// Mitsubishi GX Works2 project: 14   PLC: FX2N/FX2NC

PROGRAM MAIN
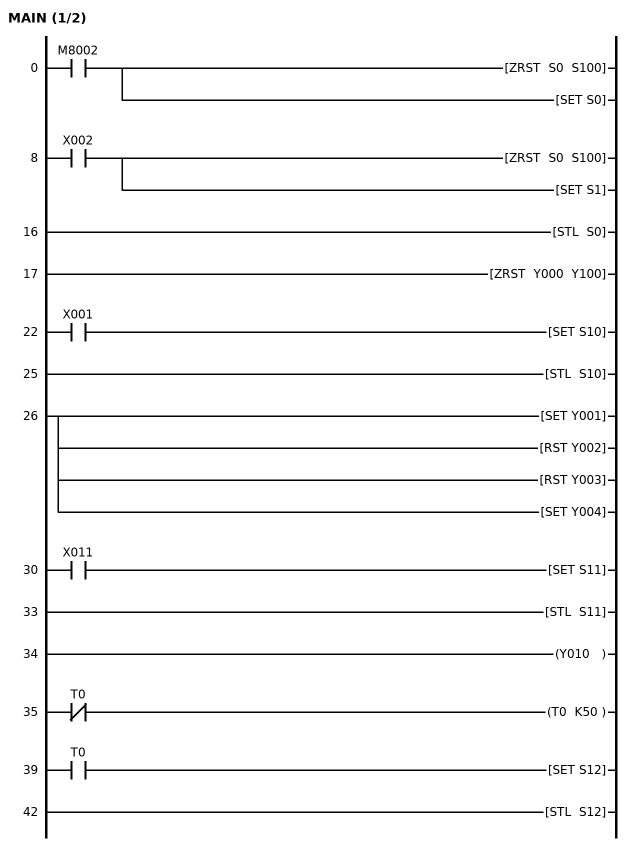
0     LD      M8002
      ZRST    S0 S100
      SET     S0
8     LD      X002
      ZRST    S0 S100
      SET     S1
16    STL     S0
17    ZRST    Y000 Y100
22    LD      X001
      SET     S10
25    STL     S10
26    SET     Y001
      RST     Y002
      RST     Y003
      SET     Y004
30    LD      X011
      SET     S11
33    STL     S11
34    OUT     Y010
35    LDI     T0
      OUT     T0 K50
39    LD      T0
      SET     S12
42    STL     S12
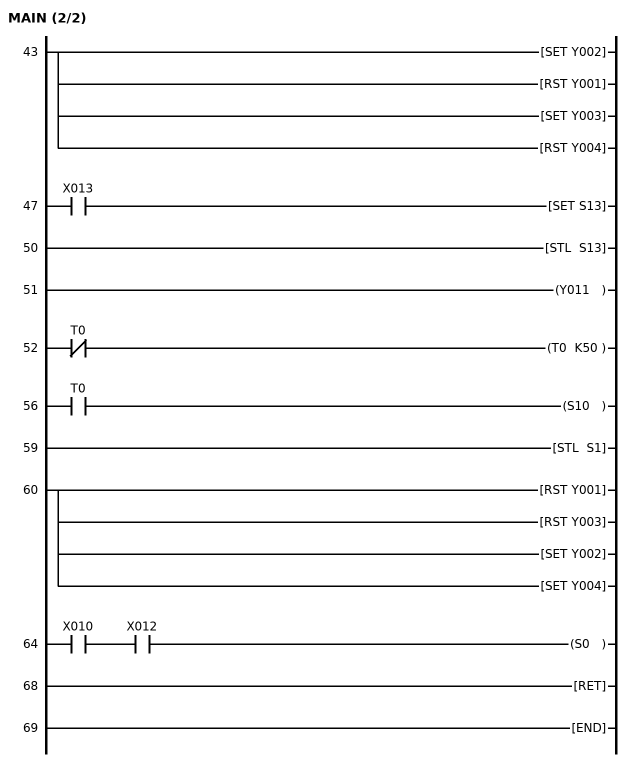
43    SET     Y002
      RST     Y001
      SET     Y003
      RST     Y004
47    LD      X013
      SET     S13
50    STL     S13
51    OUT     Y011
52    LDI     T0
      OUT     T0 K50
56    LD      T0
      OUT     S10
59    STL     S1
60    RST     Y001
      RST     Y003
      SET     Y002
      SET     Y004
64    LD      X010
      AND     X012
      OUT     S0
68    RET
69    END
END_PROGRAM

// device comments not shown above
BL0  ; main
BL1  ; a
BL2  ; b
